{attribute 'qualified_only'}
{attribute 'strict'}
TYPE E_FootpedalPos :
(
	eReverse2 	,
	eReverse1 	,
	eIdle		,
	eForward1	,
	eForward2	,
	eForward3	,
	eForward4	,
	eForward5	,
	eForward6	,
	eForward7	,
	eForward8	,
	eForward9	,
	eForward10	,
	eForward11	,
	eForward12	,
	eForward13	,
	eFalse			
) INT; 
END_TYPE

(* stored: Version 1.1.0.1, ProductVersion 3.1.4024.3
   EnumerationTextList E_FootpedalPos: Id {a45d04ff-12cb-4fd2-8aee-f6a35d915e0d} *)
